Staubli VAL3: onF5Event.pgx

program onF5Event()
  local num i
  local num l_nValue
  local string l_sMessage
begin
  // look if the bButton is enable
  if bButton[4]
    //
    call selectType()
    //
    call buildList()
    //
    use:bUseRefresh=true
  endIf
end
